(* CoDeSys 2.3.9.37 project: Cap12_7.pro *)
(* Libraries: Util.lib 18.5.10 16:14:28, Standard.lib 4.10.05 12:14:46, IecSfc.lib 13.4.06 16:51:28 *)

(* Global variable list: Global_Variables *)
VAR_GLOBAL
   (* Entradas PLC *)
   IW1_Posicion : WORD;   (* Posición rel de la valvula *)
   IX2_Error : BOOL;         (* Error en la Válvula *)
  (* Variables para el control de la visualización *)
  (* Panel de control de la valvula 1*)
   Man : BOOL;  (* Manual/Automarico *)
   RefManual : REAL;  (* SP Manual *)

   (*Salidas *)
   QW1_SPPosicion : WORD;  (* Consigna de posición para la válvula *)

(*-----------------------------------------------------*)

(* Otras variables  de la simulación*)
   QX3_ValvulaONOFF: BOOL; (* Apertura cierre válvula ON/OFF *)

END_VAR

(* POU PLC_PRG, ST *)
PROGRAM PLC_PRG
VAR
END_VAR
 ProcesoValvula();
 ProgramaControl();
END_PROGRAM

(* POU ProcesoValvula, ST *)
PROGRAM ProcesoValvula
VAR
       K: REAL :=1;
       tau : REAL:=1000;
	tact: TIME;
	tactw: DWORD;
	tinc: REAL;
	toldw: DWORD;
	Salida: REAL;
	Entrada: REAL ;
       Ciclo1:BOOL:=TRUE;
	EscalaSalida: Escalado;
	IW1R: REAL;
	EscalaEntrada: Escalado;
	QW1R: REAL;
END_VAR
  QW1R:=WORD_TO_REAL(QW1_SPPosicion);
  EscalaEntrada(Valor_Ent:=QW1R,Min_Ent:=0,Max_Ent:=4095,Min_Sal:=0,Max_Sal:=100,Valor_Sal=>Entrada);

(* Programa que simula un sistema de primer orden *)
    tact:=TIME();
    tactw:=TIME_TO_DWORD(tact);
    (* Calcula el intervalo de tiempo desde el último ciclo en milisegundos *)
    tinc:=DWORD_TO_REAL(tactw-toldw);
    (* Almacena el valor actual para al próximo ciclo *)
    toldw:=tactw;
    IF Ciclo1=FALSE THEN
        Salida:=Salida+tinc*(K*Entrada-Salida)/tau;
    ELSE
        Ciclo1:=FALSE;
    END_IF

    EscalaSalida(Valor_Ent:=Salida,Min_Ent:=0,Max_Ent:=100,Min_Sal:=0,Max_Sal:=4095,Valor_Sal=>IW1R);
    IW1_Posicion:=REAL_TO_WORD(IW1R);
END_PROGRAM

(* POU Escalado, ST *)
FUNCTION_BLOCK Escalado
VAR_INPUT
	Valor_Ent : REAL;    (* Valor a convertir *)
	Min_Ent : REAL;      (* Valor mínimo de la entrada *)
	Max_Ent : REAL;	  (* Valor máximo de la entrada *)
	Min_Sal : REAL;      (* Valor mínimo de la salida *)
	Max_Sal : REAL;	   (* . Valor máximo de la salida. *)
       ValError : REAL:=-1;    (*Valor al que poner la salida en caso de error *)
END_VAR
VAR_OUTPUT
	Valor_Sal : REAL;   (*. Valor convertido *)
	Error :  BOOL;         (* Se activa cuando el valor de entrada queda fuera de límites *)
END_VAR
VAR
	pendiente: REAL;
END_VAR
Error:= (Valor_Ent>Max_Ent) OR (Valor_Ent<Min_Ent);

IF NOT Error THEN
   pendiente:=(Max_Sal-Min_Sal)/(Max_Ent-Min_Ent);
   Valor_Sal:=Valor_Ent*pendiente+Min_Sal;
ELSE
   Valor_Sal:=ValError;
END_IF
END_FUNCTION_BLOCK

(* POU ControlValvula, ST *)
FUNCTION_BLOCK ControlValvula
VAR_INPUT
    Manual : BOOL;
    SPManual : REAL;
    SPAuto : REAL;
    PV : REAL;
    ErrorValvula : BOOL;
    SPError : REAL;
     Encl : BOOL;
     SPEncl : REAL;
END_VAR
VAR_OUTPUT
      SP:REAL;
      DIF : REAL;
      Alarma : BOOL;
END_VAR
VAR
END_VAR

END_FUNCTION_BLOCK

(* POU SenalAuto, FBD *)
FUNCTION_BLOCK SenalAuto
VAR_INPUT
END_VAR
VAR_OUTPUT
   Senal : REAL;

END_VAR
VAR
	Tempo: TON;
	STempo: BOOL;
        Salida:BOOL;
END_VAR
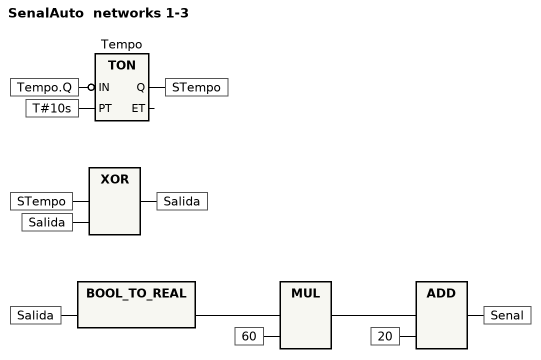
_FBD_ (* Function Block Diagram *)
NETWORK 1
	Tempo:TON(IN: NOT Tempo.Q, PT: T#10s) => STempo
NETWORK 2
	XOR(STempo, Salida) => Salida
NETWORK 3
	ADD(MUL(BOOL_TO_REAL(Salida), 60), 20) => Senal
_END_FBD_
(* the same logic as Structured Text *)
(* Network 1 *)
Tempo(IN := NOT Tempo.Q, PT := T#10s);
STempo := Tempo.Q;
(* Network 2 *)
Salida := STempo XOR Salida;
(* Network 3 *)
Senal := (BOOL_TO_REAL(Salida) * 60) + 20;
END_FUNCTION_BLOCK

(* Visualisation Visu
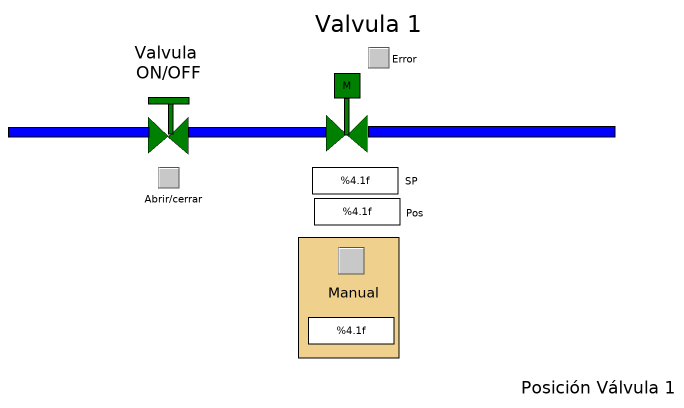
button at (490,260)-(516,287): toggles Man
rectangle at (460,330)-(546,357): text "%4.1f"; shows RefManual; editable 0..100
polygon at (478,128)-(499,164): alarm colour if IX2_Error
polygon at (499,128)-(519,165): alarm colour if IX2_Error
rectangle at (486,86)-(512,111): text "M"; alarm colour if IX2_Error
rectangle at (496,111)-(501,148): alarm colour if IX2_Error
rectangle at (464,180)-(550,207): text "%4.1f"; shows ProcesoValvula.Entrada
rectangle at (547,182)-(580,206): text "SP"
rectangle at (550,214)-(583,238): text "Pos"
rectangle at (480,290)-(531,321): text "Manual"
rectangle at (466,211)-(552,238): text "%4.1f"; shows ProcesoValvula.Salida
button at (520,60)-(541,81): toggles IX2_Error
rectangle at (540,60)-(573,84): text "Error"
rectangle at (460,20)-(581,54): text "Valvula 1"
polygon at (320,130)-(340,167): alarm colour if QX3_ValvulaONOFF
polygon at (300,130)-(321,166): alarm colour if QX3_ValvulaONOFF
rectangle at (320,110)-(325,147): alarm colour if QX3_ValvulaONOFF
rectangle at (300,110)-(341,117): alarm colour if QX3_ValvulaONOFF
rectangle at (260,50)-(381,101): text "Valvula / ON/OFF"
button at (310,180)-(331,201): toggles QX3_ValvulaONOFF
rectangle at (290,200)-(361,224): text "Abrir/cerrar"
rectangle at (670,380)-(831,421): text "Posición Válvula 1"
4 more shapes without text or variables
1 elements of other kinds (tables, trends, ...) not read
*)
